FUNCTION_BLOCK AxNcPTP EXTENDS AxNcBase implements I_AxNcPTP (* See Tc2_MC2 *)
VAR_OUTPUT CONSTANT
END_VAR
VAR_INPUT
	Motion													:	AxMotion;                                        
END_VAR                           
VAR_OUTPUT                  	
END_VAR
VAR

END_VAR

	(* Axis 																*)
	(************************************************************************)

	
(********************************************************************************)
(* Call AxNcBase																*)
(********************************************************************************)
	Super^();
		
(********************************************************************************)
(* work moving ctrl 															*)
(********************************************************************************)
	Motion(rAxis := THIS^);
	errorCheck(AxBase := Motion);
	
(********************************************************************************)

METHOD PUBLIC noAction : BOOL //Return value = TRUE if busy of home and motion 
VAR_INPUT
END_VAR

Motion.Execute	:= FALSE;
Motion.JogBwd	:= FALSE;
Motion.JogFwd	:= FALSE;

NoAction 		:= 	Super^.noAction() and NOT Motion.Busy;
END_METHOD

{attribute 'monitoring' := 'call'}
PROPERTY rMotion : REFERENCE TO AxMotion
GET
rMotion REF= Motion;
END_GET
END_PROPERTY

END_FUNCTION_BLOCK

(* stored: Version 1.1.0.1, ProductVersion 3.1.4024.6
   POU AxNcPTP: Id {029282f8-0bc8-4352-aa48-cfeb8fcdebe9}, SpecialFunc None
   Method noAction: Id {4aa31de8-13f8-41da-809d-c5fabfa1225a}
   Property rMotion: Id {9acdc345-943d-4dcc-8d8d-5031734f58d4}
   Get Get: Id {6db80e0f-b7ca-4751-b5bb-2c6e7929d405} *)
